{attribute 'qualified_only'}
{attribute 'strict'}
{attribute 'to_string'}
TYPE E_OperatingState :
(
	Init,
	MoveLinAxis,
	SetPoses,
	OperatingGalvo14mm,
	OperatingGalvo10mm,
	MirrorAdjustment,
	FinishedHandling14mm,
	FinishedHandling10mm
);
END_TYPE

(* stored: Version 1.1.0.1
   DUT E_OperatingState: Id {608413fb-457d-41a2-a61b-d1fbbfb33938} *)
